// TIA Portal V17 export
// export: Created 2023-04-03T06:31:42.2859767Z, ExportSetting WithDefaults, DisplayName Totally Integrated Automation Portal, DisplayVersion V17 Update 4, DisplayName TIA Portal Openness, DisplayVersion V17 Update 4, DisplayName TIA Portal Version Control Interface, DisplayVersion V17, DisplayName STEP 7 Professional, DisplayVersion V17 Update 4, DisplayName STEP 7 Safety, DisplayVersion V17, DisplayName WinCC Professional, DisplayVersion V17 Update 4
TYPE "W_PE_Block2"
// stored: IsFailsafeCompliant false
   STRUCT
      "G8.1.1_P_Control_Mode" : Int := 0;   // 1 / 40551
      "G8.1.2_Q_Control_Mode" : Int := 0;   // 2 / 40552
      "G8.1.3_Pac_Reference" : Real := 0.0;   // 3 / 40553
      "G8.1.4_Q_Reference" : Real := 0.0;   // 8 / 40558
      "G8.1.4a_Q_Reference_1" : Real;   // 48
      "G8.1.4b_Q_reference_2" : Real;   // 49
   END_STRUCT;
END_TYPE
